// Mitsubishi GX Works2 project: z02   PLC: Q02/Q02H

PROGRAM MAIN
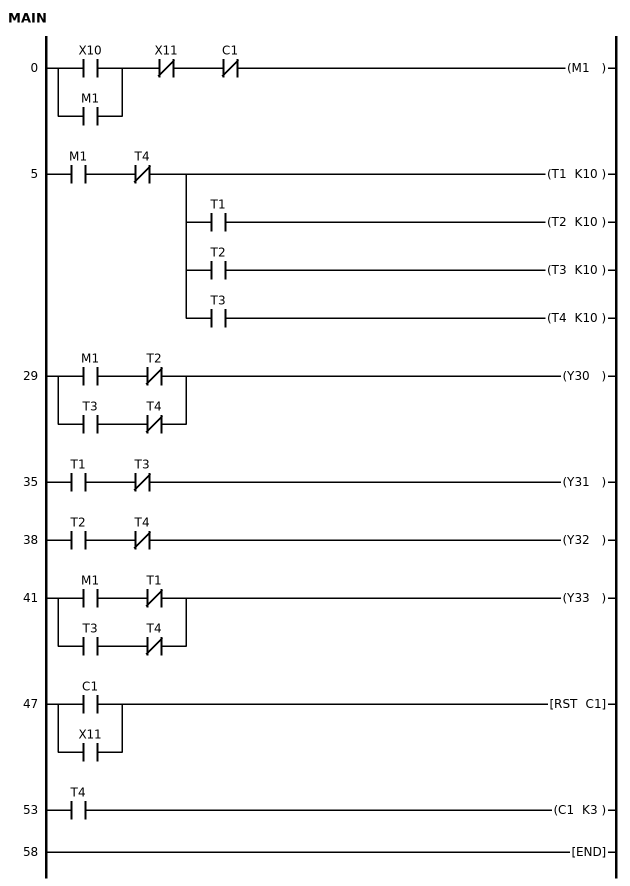
0     LD      X10
      OR      M1
      ANI     X11
      ANI     C1
      OUT     M1
5     LD      M1
      ANI     T4
      OUT     T1 K10
      MPS
      AND     T1
      OUT     T2 K10
      MRD
      AND     T2
      OUT     T3 K10
      MPP
      AND     T3
      OUT     T4 K10
29    LD      M1
      ANI     T2
      LD      T3
      ANI     T4
      ORB
      OUT     Y30
35    LD      T1
      ANI     T3
      OUT     Y31
38    LD      T2
      ANI     T4
      OUT     Y32
41    LD      M1
      ANI     T1
      LD      T3
      ANI     T4
      ORB
      OUT     Y33
47    LD      C1
      OR      X11
      RST     C1
53    LD      T4
      OUT     C1 K3
58    END
END_PROGRAM
